INTERFACE I_AlarmAddedEvent EXTENDS I_Event

PROPERTY PUBLIC Target : I_Alarm
GET
END_GET
END_PROPERTY

END_INTERFACE

(* stored: Version 1.1.0.1, ProductVersion 3.1.4024.12
   Itf I_AlarmAddedEvent: Id {a6b5112b-3551-45ae-9087-dc89dbec17ce}
   Property Target: Id {1f1ed65f-ea1c-4350-9e16-a5e26cc872a7}
   Get Get: Id {449f5696-3e87-4871-80ab-e5ce05be5033} *)
